KUKA KRL program: MasterReference.src, MasterReference.dat

--- MasterReference.src ---
&ACCESS RVP
&REL 1
&COMMENT MASTERING TEST
&PARAM EDITMASK = *
DEF MasterReference( )
;FOLD INI
  ;FOLD BASISTECH INI
    GLOBAL INTERRUPT DECL 3 WHEN $STOPMESS==TRUE DO IR_STOPM ( )
    INTERRUPT ON 3
    BAS (#INITMOV,0 )
  ;ENDFOLD (BASISTECH INI)
  ;FOLD USER INI
    ;Make your modifications here

  ;ENDFOLD (USER INI)
;ENDFOLD (INI)

  ;******************************;
  ;         TESLA MOTORS         ;
  ;ALL MODELS                    ;
  ;Program 09                    ;
  ;KUKA SAFE Program             ;
  ;Template    KRC4.V7.1         ;
  ;******************************;

MasRef_Main()


END

--- MasterReference.dat ---
&ACCESS RVP
&REL 1
&COMMENT MASTERING TEST
&PARAM EDITMASK = *
DEFDAT MasterReference
;FOLD EXTERNAL DECLARATIONS;%{PE}%MKUKATPBASIS,%CEXT,%VCOMMON,%P
;FOLD BASISTECH EXT;%{PE}%MKUKATPBASIS,%CEXT,%VEXT,%P
EXT  BAS (BAS_COMMAND  :IN,REAL  :IN )
DECL INT SUCCESS
;ENDFOLD (BASISTECH EXT)
;FOLD USER EXT;%{E}%MKUKATPUSER,%CEXT,%VEXT,%P
;Make here your modifications

;ENDFOLD (USER EXT)
;ENDFOLD (EXTERNAL DECLARATIONS)
ENDDAT
